ABB RAPID module: P702.mod

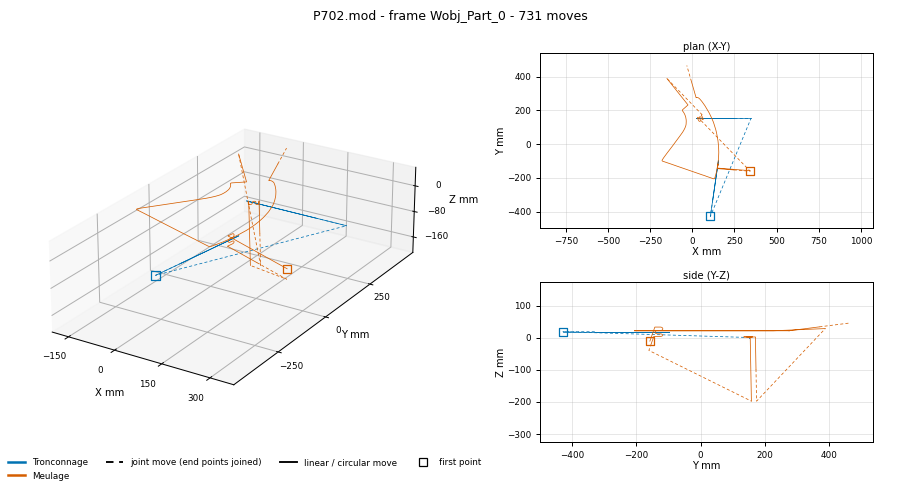
[picture p0: tool path of P702.mod in frame Wobj_Part_0, 731 of 741 moves have a stored position in this frame; points joined in program order, loops and branches not executed]
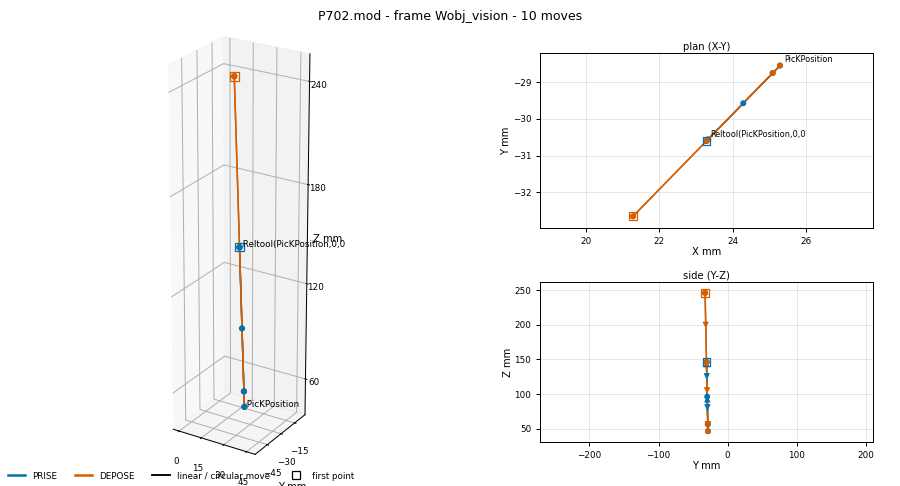
[picture p1: tool path of P702.mod in frame Wobj_vision, 10 of 741 moves have a stored position in this frame; points joined in program order, loops and branches not executed]
MODULE P702

    ! Nom         :P702
    ! Description :
    ! Créé le     :26/05/2023 11:39:24

    LOCAL CONST SPEEDDATA VitesseLente :=[10,500,0,0];
	LOCAL CONST SPEEDDATA VitesseRapide :=[30,500,0,0];
	LOCAL CONST SPEEDDATA VitesseTronconnage :=[2,500,0,0];
	LOCAL CONST SPEEDDATA VitesseTronconnageApp :=[10,500,0,0];
    !
    !Point de prise
    LOCAL PERS Robtarget PicKPosition := [[25.2898814792726,-28.5440039905978,46.3111401766051],[0.0100988844033144,-0.999721568162291,-0.0187160658859885,-0.0102228940466498],[0,0,0,0],[8.999999E+09,8.999999E+09,8.999999E+09,8.999999E+09,8.999999E+09,8.999999E+09]];
	LOCAL PERS Pose Ref := [[0,0,0],[1,0,0,0]];
    !
    !Declaration des points de meulage

    !Tr_meulage_motif_1 : Meulage d'un motif
    LOCAL CONST Robtarget Tr_meulage_motif_1_0 := [[148.038015625,-142.293734375,33.02674609375],[0.573441761718492,-0.459065341021942,-0.424059487360605,0.529714177428792],[0,0,0,0],[8.999999E+09,8.999999E+09,8.999999E+09,8.999999E+09,8.999999E+09,8.999999E+09]];
    LOCAL CONST Robtarget Tr_meulage_motif_1_1 := [[148.1818125,-141.304125,33.02651953125],[0.573441761718492,-0.459065341021942,-0.424059487360605,0.529714177428792],[0,0,0,0],[8.999999E+09,8.999999E+09,8.999999E+09,8.999999E+09,8.999999E+09,8.999999E+09]];
    LOCAL CONST Robtarget Tr_meulage_motif_1_2 := [[148.325609375,-140.314515625,33.0262890625],[0.573441761718492,-0.459065341021942,-0.424059487360605,0.529714177428792],[0,0,0,0],[8.999999E+09,8.999999E+09,8.999999E+09,8.999999E+09,8.999999E+09,8.999999E+09]];
    LOCAL CONST Robtarget Tr_meulage_motif_1_3 := [[148.46940625,-139.32490625,33.02605859375],[0.573441761718492,-0.459065341021942,-0.424059487360605,0.529714177428792],[0,0,0,0],[8.999999E+09,8.999999E+09,8.999999E+09,8.999999E+09,8.999999E+09,8.999999E+09]];
    LOCAL CONST Robtarget Tr_meulage_motif_1_4 := [[148.613203125,-138.335296875,33.025828125],[0.573441761718492,-0.459065341021942,-0.424059487360605,0.529714177428792],[0,0,0,0],[8.999999E+09,8.999999E+09,8.999999E+09,8.999999E+09,8.999999E+09,8.999999E+09]];
    LOCAL CONST Robtarget Tr_meulage_motif_1_5 := [[148.757,-137.3456875,33.02559765625],[0.573441761718492,-0.459065341021942,-0.424059487360605,0.529714177428792],[0,0,0,0],[8.999999E+09,8.999999E+09,8.999999E+09,8.999999E+09,8.999999E+09,8.999999E+09]];
    LOCAL CONST Robtarget Tr_meulage_motif_1_6 := [[148.900796875,-136.35609375,33.0253671875],[0.573441761718492,-0.459065341021942,-0.424059487360605,0.529714177428792],[0,0,0,0],[8.999999E+09,8.999999E+09,8.999999E+09,8.999999E+09,8.999999E+09,8.999999E+09]];
    LOCAL CONST Robtarget Tr_meulage_motif_1_7 := [[149.04459375,-135.366484375,33.02513671875],[0.573441761718492,-0.459065341021942,-0.424059487360605,0.529714177428792],[0,0,0,0],[8.999999E+09,8.999999E+09,8.999999E+09,8.999999E+09,8.999999E+09,8.999999E+09]];
    LOCAL CONST Robtarget Tr_meulage_motif_1_8 := [[149.188390625,-134.376875,33.02490625],[0.573441761718492,-0.459065341021942,-0.424059487360605,0.529714177428792],[0,0,0,0],[8.999999E+09,8.999999E+09,8.999999E+09,8.999999E+09,8.999999E+09,8.999999E+09]];
    LOCAL CONST Robtarget Tr_meulage_motif_1_9 := [[149.3321875,-133.387265625,33.02467578125],[0.573441761718492,-0.459065341021942,-0.424059487360605,0.529714177428792],[0,0,0,0],[8.999999E+09,8.999999E+09,8.999999E+09,8.999999E+09,8.999999E+09,8.999999E+09]];
    LOCAL CONST Robtarget Tr_meulage_motif_1_10 := [[149.475984375,-132.39765625,33.0244453125],[0.573441761718492,-0.459065341021942,-0.424059487360605,0.529714177428792],[0,0,0,0],[8.999999E+09,8.999999E+09,8.999999E+09,8.999999E+09,8.999999E+09,8.999999E+09]];
    LOCAL CONST Robtarget Tr_meulage_motif_1_11 := [[149.61978125,-131.408046875,33.02421484375],[0.573441761718492,-0.459065341021942,-0.424059487360605,0.529714177428792],[0,0,0,0],[8.999999E+09,8.999999E+09,8.999999E+09,8.999999E+09,8.999999E+09,8.999999E+09]];
    LOCAL CONST Robtarget Tr_meulage_motif_1_12 := [[149.763578125,-130.4184453125,33.023984375],[0.573441761718492,-0.459065341021942,-0.424059487360605,0.529714177428792],[0,0,0,0],[8.999999E+09,8.999999E+09,8.999999E+09,8.999999E+09,8.999999E+09,8.999999E+09]];
    LOCAL CONST Robtarget Tr_meulage_motif_1_13 := [[149.907375,-129.4288359375,33.0237578125],[0.573441761718492,-0.459065341021942,-0.424059487360605,0.529714177428792],[0,0,0,0],[8.999999E+09,8.999999E+09,8.999999E+09,8.999999E+09,8.999999E+09,8.999999E+09]];
    LOCAL CONST Robtarget Tr_meulage_motif_1_14 := [[150.051171875,-128.4392265625,33.02352734375],[0.573441761718492,-0.459065341021942,-0.424059487360605,0.529714177428792],[0,0,0,0],[8.999999E+09,8.999999E+09,8.999999E+09,8.999999E+09,8.999999E+09,8.999999E+09]];
    LOCAL CONST Robtarget Tr_meulage_motif_1_15 := [[150.19496875,-127.449625,33.023296875],[0.573441761718492,-0.459065341021942,-0.424059487360605,0.529714177428792],[0,0,0,0],[8.999999E+09,8.999999E+09,8.999999E+09,8.999999E+09,8.999999E+09,8.999999E+09]];
    LOCAL CONST Robtarget Tr_meulage_motif_1_16 := [[150.338765625,-126.460015625,33.02306640625],[0.573441761718492,-0.459065341021942,-0.424059487360605,0.529714177428792],[0,0,0,0],[8.999999E+09,8.999999E+09,8.999999E+09,8.999999E+09,8.999999E+09,8.999999E+09]];
    LOCAL CONST Robtarget Tr_meulage_motif_1_17 := [[150.4825625,-125.47040625,33.0228359375],[0.573441761718492,-0.459065341021942,-0.424059487360605,0.529714177428792],[0,0,0,0],[8.999999E+09,8.999999E+09,8.999999E+09,8.999999E+09,8.999999E+09,8.999999E+09]];
    LOCAL CONST Robtarget Tr_meulage_motif_1_18 := [[150.626359375,-124.480796875,33.02260546875],[0.573441761718492,-0.459065341021942,-0.424059487360605,0.529714177428792],[0,0,0,0],[8.999999E+09,8.999999E+09,8.999999E+09,8.999999E+09,8.999999E+09,8.999999E+09]];
    LOCAL CONST Robtarget Tr_meulage_motif_1_19 := [[150.7724375,-123.4990703125,32.9118359375],[0.573441761718492,-0.459065341021942,-0.424059487360605,0.529714177428792],[0,0,0,0],[8.999999E+09,8.999999E+09,8.999999E+09,8.999999E+09,8.999999E+09,8.999999E+09]];
    LOCAL CONST Robtarget Tr_meulage_motif_1_20 := [[150.914953125,-122.5633828125,32.700529296875],[0.573441761718492,-0.459065341021942,-0.424059487360605,0.529714177428792],[0,0,0,0],[8.999999E+09,8.999999E+09,8.999999E+09,8.999999E+09,8.999999E+09,8.999999E+09]];
    LOCAL CONST Robtarget Tr_meulage_motif_1_21 := [[151.045796875,-121.7207890625,32.4286171875],[0.573441761718492,-0.459065341021942,-0.424059487360605,0.529714177428792],[0,0,0,0],[8.999999E+09,8.999999E+09,8.999999E+09,8.999999E+09,8.999999E+09,8.999999E+09]];
    LOCAL CONST Robtarget Tr_meulage_motif_1_22 := [[151.162,-120.979921875,32.15263671875],[0.573441761718492,-0.459065341021942,-0.424059487360605,0.529714177428792],[0,0,0,0],[8.999999E+09,8.999999E+09,8.999999E+09,8.999999E+09,8.999999E+09,8.999999E+09]];
    LOCAL CONST Robtarget Tr_meulage_motif_1_23 := [[151.339015625,-119.89315625,31.536548828125],[0.573441761718492,-0.459065341021942,-0.424059487360605,0.529714177428792],[0,0,0,0],[8.999999E+09,8.999999E+09,8.999999E+09,8.999999E+09,8.999999E+09,8.999999E+09]];
    LOCAL CONST Robtarget Tr_meulage_motif_1_24 := [[151.5119375,-118.883859375,30.6890546875],[0.573441761718492,-0.459065341021942,-0.424059487360605,0.529714177428792],[0,0,0,0],[8.999999E+09,8.999999E+09,8.999999E+09,8.999999E+09,8.999999E+09,8.999999E+09]];
    LOCAL CONST Robtarget Tr_meulage_motif_1_25 := [[151.664859375,-118.0497578125,29.665466796875],[0.573441761718492,-0.459065341021942,-0.424059487360605,0.529714177428792],[0,0,0,0],[8.999999E+09,8.999999E+09,8.999999E+09,8.999999E+09,8.999999E+09,8.999999E+09]];
    LOCAL CONST Robtarget Tr_meulage_motif_1_26 := [[151.768890625,-117.5718515625,28.54969140625],[0.573441761718492,-0.459065341021942,-0.424059487360605,0.529714177428792],[0,0,0,0],[8.999999E+09,8.999999E+09,8.999999E+09,8.999999E+09,8.999999E+09,8.999999E+09]];
    LOCAL CONST Robtarget Tr_meulage_motif_1_27 := [[151.793875,-117.548296875,27.85404296875],[0.573441761718492,-0.459065341021942,-0.424059487360605,0.529714177428792],[0,0,0,0],[8.999999E+09,8.999999E+09,8.999999E+09,8.999999E+09,8.999999E+09,8.999999E+09]];
    LOCAL CONST Robtarget Tr_meulage_motif_1_28 := [[151.813921875,-117.551359375,27.193103515625],[0.573441761718492,-0.459065341021942,-0.424059487360605,0.529714177428792],[0,0,0,0],[8.999999E+09,8.999999E+09,8.999999E+09,8.999999E+09,8.999999E+09,8.999999E+09]];
    LOCAL CONST Robtarget Tr_meulage_motif_1_29 := [[151.8260625,-117.608734375,26.532333984375],[0.573441761718492,-0.459065341021942,-0.424059487360605,0.529714177428792],[0,0,0,0],[8.999999E+09,8.999999E+09,8.999999E+09,8.999999E+09,8.999999E+09,8.999999E+09]];
    LOCAL CONST Robtarget Tr_meulage_motif_1_30 := [[151.7878125,-118.1068828125,25.431216796875],[0.573441761718492,-0.459065341021942,-0.424059487360605,0.529714177428792],[0,0,0,0],[8.999999E+09,8.999999E+09,8.999999E+09,8.999999E+09,8.999999E+09,8.999999E+09]];
    LOCAL CONST Robtarget Tr_meulage_motif_1_31 := [[151.695140625,-118.9592734375,24.42526171875],[0.573441761718492,-0.459065341021942,-0.424059487360605,0.529714177428792],[0,0,0,0],[8.999999E+09,8.999999E+09,8.999999E+09,8.999999E+09,8.999999E+09,8.999999E+09]];
    LOCAL CONST Robtarget Tr_meulage_motif_1_32 := [[151.573109375,-119.9758828125,23.59701171875],[0.573441761718492,-0.459065341021942,-0.424059487360605,0.529714177428792],[0,0,0,0],[8.999999E+09,8.999999E+09,8.999999E+09,8.999999E+09,8.999999E+09,8.999999E+09]];
    LOCAL CONST Robtarget Tr_meulage_motif_1_33 := [[151.486296875,-120.657671875,23.201607421875],[0.573441761718492,-0.459065341021942,-0.424059487360605,0.529714177428792],[0,0,0,0],[8.999999E+09,8.999999E+09,8.999999E+09,8.999999E+09,8.999999E+09,8.999999E+09]];
    LOCAL CONST Robtarget Tr_meulage_motif_1_34 := [[151.33453125,-121.8060546875,22.714572265625],[0.573441761718492,-0.459065341021942,-0.424059487360605,0.529714177428792],[0,0,0,0],[8.999999E+09,8.999999E+09,8.999999E+09,8.999999E+09,8.999999E+09,8.999999E+09]];
    LOCAL CONST Robtarget Tr_meulage_motif_1_35 := [[151.22103125,-122.6435234375,22.450796875],[0.573441761718492,-0.459065341021942,-0.424059487360605,0.529714177428792],[0,0,0,0],[8.999999E+09,8.999999E+09,8.999999E+09,8.999999E+09,8.999999E+09,8.999999E+09]];
    LOCAL CONST Robtarget Tr_meulage_motif_1_36 := [[151.093203125,-123.5667890625,22.246638671875],[0.573441761718492,-0.459065341021942,-0.424059487360605,0.529714177428792],[0,0,0,0],[8.999999E+09,8.999999E+09,8.999999E+09,8.999999E+09,8.999999E+09,8.999999E+09]];
    LOCAL CONST Robtarget Tr_meulage_motif_1_37 := [[150.955359375,-124.53865625,22.138322265625],[0.573441761718492,-0.459065341021942,-0.424059487360605,0.529714177428792],[0,0,0,0],[8.999999E+09,8.999999E+09,8.999999E+09,8.999999E+09,8.999999E+09,8.999999E+09]];
    LOCAL CONST Robtarget Tr_meulage_motif_1_38 := [[150.815984375,-125.5214140625,22.0280078125],[0.573441761718492,-0.459065341021942,-0.424059487360605,0.529714177428792],[0,0,0,0],[8.999999E+09,8.999999E+09,8.999999E+09,8.999999E+09,8.999999E+09,8.999999E+09]];
    LOCAL CONST Robtarget Tr_meulage_motif_1_39 := [[150.6721875,-126.511015625,22.02823828125],[0.573441761718492,-0.459065341021942,-0.424059487360605,0.529714177428792],[0,0,0,0],[8.999999E+09,8.999999E+09,8.999999E+09,8.999999E+09,8.999999E+09,8.999999E+09]];
    LOCAL CONST Robtarget Tr_meulage_motif_1_40 := [[150.528390625,-127.500625,22.02846875],[0.573441761718492,-0.459065341021942,-0.424059487360605,0.529714177428792],[0,0,0,0],[8.999999E+09,8.999999E+09,8.999999E+09,8.999999E+09,8.999999E+09,8.999999E+09]];
    LOCAL CONST Robtarget Tr_meulage_motif_1_41 := [[150.38459375,-128.490234375,22.02869921875],[0.573441761718492,-0.459065341021942,-0.424059487360605,0.529714177428792],[0,0,0,0],[8.999999E+09,8.999999E+09,8.999999E+09,8.999999E+09,8.999999E+09,8.999999E+09]];
    LOCAL CONST Robtarget Tr_meulage_motif_1_42 := [[150.240796875,-129.47984375,22.028927734375],[0.573441761718492,-0.459065341021942,-0.424059487360605,0.529714177428792],[0,0,0,0],[8.999999E+09,8.999999E+09,8.999999E+09,8.999999E+09,8.999999E+09,8.999999E+09]];
    LOCAL CONST Robtarget Tr_meulage_motif_1_43 := [[150.097,-130.4694453125,22.029158203125],[0.573441761718492,-0.459065341021942,-0.424059487360605,0.529714177428792],[0,0,0,0],[8.999999E+09,8.999999E+09,8.999999E+09,8.999999E+09,8.999999E+09,8.999999E+09]];
    LOCAL CONST Robtarget Tr_meulage_motif_1_44 := [[149.953203125,-131.4590625,22.029388671875],[0.573441761718492,-0.459065341021942,-0.424059487360605,0.529714177428792],[0,0,0,0],[8.999999E+09,8.999999E+09,8.999999E+09,8.999999E+09,8.999999E+09,8.999999E+09]];
    LOCAL CONST Robtarget Tr_meulage_motif_1_45 := [[149.80940625,-132.44865625,22.029619140625],[0.573441761718492,-0.459065341021942,-0.424059487360605,0.529714177428792],[0,0,0,0],[8.999999E+09,8.999999E+09,8.999999E+09,8.999999E+09,8.999999E+09,8.999999E+09]];
    LOCAL CONST Robtarget Tr_meulage_motif_1_46 := [[149.665609375,-133.438265625,22.029849609375],[0.573441761718492,-0.459065341021942,-0.424059487360605,0.529714177428792],[0,0,0,0],[8.999999E+09,8.999999E+09,8.999999E+09,8.999999E+09,8.999999E+09,8.999999E+09]];
    LOCAL CONST Robtarget Tr_meulage_motif_1_47 := [[149.5218125,-134.427875,22.030080078125],[0.573441761718492,-0.459065341021942,-0.424059487360605,0.529714177428792],[0,0,0,0],[8.999999E+09,8.999999E+09,8.999999E+09,8.999999E+09,8.999999E+09,8.999999E+09]];
    LOCAL CONST Robtarget Tr_meulage_motif_1_48 := [[149.378015625,-135.417484375,22.03030859375],[0.573441761718492,-0.459065341021942,-0.424059487360605,0.529714177428792],[0,0,0,0],[8.999999E+09,8.999999E+09,8.999999E+09,8.999999E+09,8.999999E+09,8.999999E+09]];
    LOCAL CONST Robtarget Tr_meulage_motif_1_49 := [[149.238640625,-136.40025,21.91999609375],[0.573441761718492,-0.459065341021942,-0.424059487360605,0.529714177428792],[0,0,0,0],[8.999999E+09,8.999999E+09,8.999999E+09,8.999999E+09,8.999999E+09,8.999999E+09]];
    LOCAL CONST Robtarget Tr_meulage_motif_1_50 := [[149.1089375,-137.337890625,21.709125],[0.573441761718492,-0.459065341021942,-0.424059487360605,0.529714177428792],[0,0,0,0],[8.999999E+09,8.999999E+09,8.999999E+09,8.999999E+09,8.999999E+09,8.999999E+09]];
    LOCAL CONST Robtarget Tr_meulage_motif_1_51 := [[148.994546875,-138.183,21.43760546875],[0.573441761718492,-0.459065341021942,-0.424059487360605,0.529714177428792],[0,0,0,0],[8.999999E+09,8.999999E+09,8.999999E+09,8.999999E+09,8.999999E+09,8.999999E+09]];
    LOCAL CONST Robtarget Tr_meulage_motif_1_52 := [[148.90146875,-138.888515625,21.133755859375],[0.573441761718492,-0.459065341021942,-0.424059487360605,0.529714177428792],[0,0,0,0],[8.999999E+09,8.999999E+09,8.999999E+09,8.999999E+09,8.999999E+09,8.999999E+09]];
    LOCAL CONST Robtarget Tr_meulage_motif_1_53 := [[148.772796875,-139.9153125,20.471775390625],[0.573441761718492,-0.459065341021942,-0.424059487360605,0.529714177428792],[0,0,0,0],[8.999999E+09,8.999999E+09,8.999999E+09,8.999999E+09,8.999999E+09,8.999999E+09]];
    LOCAL CONST Robtarget Tr_meulage_motif_1_54 := [[148.6704375,-140.8120625,19.57046875],[0.573441761718492,-0.459065341021942,-0.424059487360605,0.529714177428792],[0,0,0,0],[8.999999E+09,8.999999E+09,8.999999E+09,8.999999E+09,8.999999E+09,8.999999E+09]];
    LOCAL CONST Robtarget Tr_meulage_motif_1_55 := [[148.62521875,-141.3463125,18.525052734375],[0.573441761718492,-0.459065341021942,-0.424059487360605,0.529714177428792],[0,0,0,0],[8.999999E+09,8.999999E+09,8.999999E+09,8.999999E+09,8.999999E+09,8.999999E+09]];
    LOCAL CONST Robtarget Tr_meulage_motif_1_56 := [[148.61965625,-141.532390625,17.832203125],[0.573441761718492,-0.459065341021942,-0.424059487360605,0.529714177428792],[0,0,0,0],[8.999999E+09,8.999999E+09,8.999999E+09,8.999999E+09,8.999999E+09,8.999999E+09]];
    LOCAL CONST Robtarget Tr_meulage_motif_1_57 := [[148.6338125,-141.599140625,17.062580078125],[0.573441761718492,-0.459065341021942,-0.424059487360605,0.529714177428792],[0,0,0,0],[8.999999E+09,8.999999E+09,8.999999E+09,8.999999E+09,8.999999E+09,8.999999E+09]];
    LOCAL CONST Robtarget Tr_meulage_motif_1_58 := [[148.666765625,-141.53646875,16.29305078125],[0.573441761718492,-0.459065341021942,-0.424059487360605,0.529714177428792],[0,0,0,0],[8.999999E+09,8.999999E+09,8.999999E+09,8.999999E+09,8.999999E+09,8.999999E+09]];
    LOCAL CONST Robtarget Tr_meulage_motif_1_59 := [[148.760703125,-141.126375,15.1852255859375],[0.573441761718492,-0.459065341021942,-0.424059487360605,0.529714177428792],[0,0,0,0],[8.999999E+09,8.999999E+09,8.999999E+09,8.999999E+09,8.999999E+09,8.999999E+09]];
    LOCAL CONST Robtarget Tr_meulage_motif_1_60 := [[148.83803125,-140.719078125,14.5997177734375],[0.573441761718492,-0.459065341021942,-0.424059487360605,0.529714177428792],[0,0,0,0],[8.999999E+09,8.999999E+09,8.999999E+09,8.999999E+09,8.999999E+09,8.999999E+09]];
    LOCAL CONST Robtarget Tr_meulage_motif_1_61 := [[148.992484375,-139.845296875,13.7128056640625],[0.573441761718492,-0.459065341021942,-0.424059487360605,0.529714177428792],[0,0,0,0],[8.999999E+09,8.999999E+09,8.999999E+09,8.999999E+09,8.999999E+09,8.999999E+09]];
    LOCAL CONST Robtarget Tr_meulage_motif_1_62 := [[149.089265625,-139.267609375,13.2985537109375],[0.573441761718492,-0.459065341021942,-0.424059487360605,0.529714177428792],[0,0,0,0],[8.999999E+09,8.999999E+09,8.999999E+09,8.999999E+09,8.999999E+09,8.999999E+09]];
    LOCAL CONST Robtarget Tr_meulage_motif_1_63 := [[149.2665,-138.16384375,12.7544580078125],[0.573441761718492,-0.459065341021942,-0.424059487360605,0.529714177428792],[0,0,0,0],[8.999999E+09,8.999999E+09,8.999999E+09,8.999999E+09,8.999999E+09,8.999999E+09]];
    LOCAL CONST Robtarget Tr_meulage_motif_1_64 := [[149.3941875,-137.348203125,12.4589072265625],[0.573441761718492,-0.459065341021942,-0.424059487360605,0.529714177428792],[0,0,0,0],[8.999999E+09,8.999999E+09,8.999999E+09,8.999999E+09,8.999999E+09,8.999999E+09]];
    LOCAL CONST Robtarget Tr_meulage_motif_1_65 := [[149.534390625,-136.42684375,12.2543203125],[0.573441761718492,-0.459065341021942,-0.424059487360605,0.529714177428792],[0,0,0,0],[8.999999E+09,8.999999E+09,8.999999E+09,8.999999E+09,8.999999E+09,8.999999E+09]];
    LOCAL CONST Robtarget Tr_meulage_motif_1_66 := [[149.678828125,-135.455984375,12.1455517578125],[0.573441761718492,-0.459065341021942,-0.424059487360605,0.529714177428792],[0,0,0,0],[8.999999E+09,8.999999E+09,8.999999E+09,8.999999E+09,8.999999E+09,8.999999E+09]];
    LOCAL CONST Robtarget Tr_meulage_motif_1_67 := [[149.82490625,-134.47425,12.03478125],[0.573441761718492,-0.459065341021942,-0.424059487360605,0.529714177428792],[0,0,0,0],[8.999999E+09,8.999999E+09,8.999999E+09,8.999999E+09,8.999999E+09,8.999999E+09]];
    LOCAL CONST Robtarget Tr_meulage_motif_1_68 := [[149.968703125,-133.484640625,12.0345517578125],[0.573441761718492,-0.459065341021942,-0.424059487360605,0.529714177428792],[0,0,0,0],[8.999999E+09,8.999999E+09,8.999999E+09,8.999999E+09,8.999999E+09,8.999999E+09]];
    LOCAL CONST Robtarget Tr_meulage_motif_1_69 := [[150.1125,-132.49503125,12.0343212890625],[0.573441761718492,-0.459065341021942,-0.424059487360605,0.529714177428792],[0,0,0,0],[8.999999E+09,8.999999E+09,8.999999E+09,8.999999E+09,8.999999E+09,8.999999E+09]];
    LOCAL CONST Robtarget Tr_meulage_motif_1_70 := [[150.256296875,-131.505421875,12.0340908203125],[0.573441761718492,-0.459065341021942,-0.424059487360605,0.529714177428792],[0,0,0,0],[8.999999E+09,8.999999E+09,8.999999E+09,8.999999E+09,8.999999E+09,8.999999E+09]];
    LOCAL CONST Robtarget Tr_meulage_motif_1_71 := [[150.40009375,-130.5158125,12.033861328125],[0.573441761718492,-0.459065341021942,-0.424059487360605,0.529714177428792],[0,0,0,0],[8.999999E+09,8.999999E+09,8.999999E+09,8.999999E+09,8.999999E+09,8.999999E+09]];
    LOCAL CONST Robtarget Tr_meulage_motif_1_72 := [[150.543890625,-129.5262109375,12.033630859375],[0.573441761718492,-0.459065341021942,-0.424059487360605,0.529714177428792],[0,0,0,0],[8.999999E+09,8.999999E+09,8.999999E+09,8.999999E+09,8.999999E+09,8.999999E+09]];
    LOCAL CONST Robtarget Tr_meulage_motif_1_73 := [[150.6876875,-128.5366015625,12.033400390625],[0.573441761718492,-0.459065341021942,-0.424059487360605,0.529714177428792],[0,0,0,0],[8.999999E+09,8.999999E+09,8.999999E+09,8.999999E+09,8.999999E+09,8.999999E+09]];
    LOCAL CONST Robtarget Tr_meulage_motif_1_74 := [[150.831484375,-127.5469921875,12.0331708984375],[0.573441761718492,-0.459065341021942,-0.424059487360605,0.529714177428792],[0,0,0,0],[8.999999E+09,8.999999E+09,8.999999E+09,8.999999E+09,8.999999E+09,8.999999E+09]];
    LOCAL CONST Robtarget Tr_meulage_motif_1_75 := [[150.97528125,-126.557390625,12.0329404296875],[0.573441761718492,-0.459065341021942,-0.424059487360605,0.529714177428792],[0,0,0,0],[8.999999E+09,8.999999E+09,8.999999E+09,8.999999E+09,8.999999E+09,8.999999E+09]];
    LOCAL CONST Robtarget Tr_meulage_motif_1_76 := [[151.119078125,-125.56778125,12.0327099609375],[0.573441761718492,-0.459065341021942,-0.424059487360605,0.529714177428792],[0,0,0,0],[8.999999E+09,8.999999E+09,8.999999E+09,8.999999E+09,8.999999E+09,8.999999E+09]];
    LOCAL CONST Robtarget Tr_meulage_motif_1_77 := [[151.262875,-124.578171875,12.03248046875],[0.573441761718492,-0.459065341021942,-0.424059487360605,0.529714177428792],[0,0,0,0],[8.999999E+09,8.999999E+09,8.999999E+09,8.999999E+09,8.999999E+09,8.999999E+09]];
    LOCAL CONST Robtarget Tr_meulage_motif_1_78 := [[151.40896875,-123.5964375,11.9217099609375],[0.573441761718492,-0.459065341021942,-0.424059487360605,0.529714177428792],[0,0,0,0],[8.999999E+09,8.999999E+09,8.999999E+09,8.999999E+09,8.999999E+09,8.999999E+09]];
    LOCAL CONST Robtarget Tr_meulage_motif_1_79 := [[151.55146875,-122.6607578125,11.710404296875],[0.573441761718492,-0.459065341021942,-0.424059487360605,0.529714177428792],[0,0,0,0],[8.999999E+09,8.999999E+09,8.999999E+09,8.999999E+09,8.999999E+09,8.999999E+09]];
    LOCAL CONST Robtarget Tr_meulage_motif_1_80 := [[151.682328125,-121.81815625,11.4384921875],[0.573441761718492,-0.459065341021942,-0.424059487360605,0.529714177428792],[0,0,0,0],[8.999999E+09,8.999999E+09,8.999999E+09,8.999999E+09,8.999999E+09,8.999999E+09]];
    LOCAL CONST Robtarget Tr_meulage_motif_1_81 := [[151.79853125,-121.077296875,11.16251171875],[0.573441761718492,-0.459065341021942,-0.424059487360605,0.529714177428792],[0,0,0,0],[8.999999E+09,8.999999E+09,8.999999E+09,8.999999E+09,8.999999E+09,8.999999E+09]];
    LOCAL CONST Robtarget Tr_meulage_motif_1_82 := [[151.97553125,-119.99053125,10.5464228515625],[0.573441761718492,-0.459065341021942,-0.424059487360605,0.529714177428792],[0,0,0,0],[8.999999E+09,8.999999E+09,8.999999E+09,8.999999E+09,8.999999E+09,8.999999E+09]];
    LOCAL CONST Robtarget Tr_meulage_motif_1_83 := [[152.140203125,-119.0478984375,9.652654296875],[0.573441761718492,-0.459065341021942,-0.424059487360605,0.529714177428792],[0,0,0,0],[8.999999E+09,8.999999E+09,8.999999E+09,8.999999E+09,8.999999E+09,8.999999E+09]];
    LOCAL CONST Robtarget Tr_meulage_motif_1_84 := [[152.260703125,-118.450140625,8.5670244140625],[0.573441761718492,-0.459065341021942,-0.424059487360605,0.529714177428792],[0,0,0,0],[8.999999E+09,8.999999E+09,8.999999E+09,8.999999E+09,8.999999E+09,8.999999E+09]];
    LOCAL CONST Robtarget Tr_meulage_motif_1_85 := [[152.314890625,-118.28715625,7.58307373046875],[0.573441761718492,-0.459065341021942,-0.424059487360605,0.529714177428792],[0,0,0,0],[8.999999E+09,8.999999E+09,8.999999E+09,8.999999E+09,8.999999E+09,8.999999E+09]];
    LOCAL CONST Robtarget Tr_meulage_motif_1_86 := [[152.3021875,-118.418203125,7.3785439453125],[0.573441761718492,-0.459065341021942,-0.424059487360605,0.529714177428792],[0,0,0,0],[8.999999E+09,8.999999E+09,8.999999E+09,8.999999E+09,8.999999E+09,8.999999E+09]];
    LOCAL CONST Robtarget Tr_meulage_motif_1_87 := [[152.30646875,-118.5436640625,6.6525078125],[0.573441761718492,-0.459065341021942,-0.424059487360605,0.529714177428792],[0,0,0,0],[8.999999E+09,8.999999E+09,8.999999E+09,8.999999E+09,8.999999E+09,8.999999E+09]];
    LOCAL CONST Robtarget Tr_meulage_motif_1_88 := [[152.236515625,-119.2248984375,5.71619921875],[0.573441761718492,-0.459065341021942,-0.424059487360605,0.529714177428792],[0,0,0,0],[8.999999E+09,8.999999E+09,8.999999E+09,8.999999E+09,8.999999E+09,8.999999E+09]];
    LOCAL CONST Robtarget Tr_meulage_motif_1_89 := [[152.170375,-119.7788828125,5.2527333984375],[0.573441761718492,-0.459065341021942,-0.424059487360605,0.529714177428792],[0,0,0,0],[8.999999E+09,8.999999E+09,8.999999E+09,8.999999E+09,8.999999E+09,8.999999E+09]];
    LOCAL CONST Robtarget Tr_meulage_motif_1_90 := [[152.023921875,-120.89990625,4.72280517578125],[0.573441761718492,-0.459065341021942,-0.424059487360605,0.529714177428792],[0,0,0,0],[8.999999E+09,8.999999E+09,8.999999E+09,8.999999E+09,8.999999E+09,8.999999E+09]];
    LOCAL CONST Robtarget Tr_meulage_motif_1_91 := [[151.910421875,-121.7373828125,4.4590302734375],[0.573441761718492,-0.459065341021942,-0.424059487360605,0.529714177428792],[0,0,0,0],[8.999999E+09,8.999999E+09,8.999999E+09,8.999999E+09,8.999999E+09,8.999999E+09]];
    LOCAL CONST Robtarget Tr_meulage_motif_1_92 := [[151.78259375,-122.660640625,4.2548720703125],[0.573441761718492,-0.459065341021942,-0.424059487360605,0.529714177428792],[0,0,0,0],[8.999999E+09,8.999999E+09,8.999999E+09,8.999999E+09,8.999999E+09,8.999999E+09]];
    LOCAL CONST Robtarget Tr_meulage_motif_1_93 := [[151.644734375,-123.6325078125,4.14655517578125],[0.573441761718492,-0.459065341021942,-0.424059487360605,0.529714177428792],[0,0,0,0],[8.999999E+09,8.999999E+09,8.999999E+09,8.999999E+09,8.999999E+09,8.999999E+09]];
    LOCAL CONST Robtarget Tr_meulage_motif_1_94 := [[151.505359375,-124.615265625,4.03624194335938],[0.573441761718492,-0.459065341021942,-0.424059487360605,0.529714177428792],[0,0,0,0],[8.999999E+09,8.999999E+09,8.999999E+09,8.999999E+09,8.999999E+09,8.999999E+09]];
    LOCAL CONST Robtarget Tr_meulage_motif_1_95 := [[151.3615625,-125.604875,4.03647216796875],[0.573441761718492,-0.459065341021942,-0.424059487360605,0.529714177428792],[0,0,0,0],[8.999999E+09,8.999999E+09,8.999999E+09,8.999999E+09,8.999999E+09,8.999999E+09]];
    LOCAL CONST Robtarget Tr_meulage_motif_1_96 := [[151.217765625,-126.594484375,4.0367021484375],[0.573441761718492,-0.459065341021942,-0.424059487360605,0.529714177428792],[0,0,0,0],[8.999999E+09,8.999999E+09,8.999999E+09,8.999999E+09,8.999999E+09,8.999999E+09]];
    LOCAL CONST Robtarget Tr_meulage_motif_1_97 := [[151.07396875,-127.5840859375,4.03693237304688],[0.573441761718492,-0.459065341021942,-0.424059487360605,0.529714177428792],[0,0,0,0],[8.999999E+09,8.999999E+09,8.999999E+09,8.999999E+09,8.999999E+09,8.999999E+09]];
    LOCAL CONST Robtarget Tr_meulage_motif_1_98 := [[150.930171875,-128.5736953125,4.03716259765625],[0.573441761718492,-0.459065341021942,-0.424059487360605,0.529714177428792],[0,0,0,0],[8.999999E+09,8.999999E+09,8.999999E+09,8.999999E+09,8.999999E+09,8.999999E+09]];
    LOCAL CONST Robtarget Tr_meulage_motif_1_99 := [[150.786375,-129.5633046875,4.037392578125],[0.573441761718492,-0.459065341021942,-0.424059487360605,0.529714177428792],[0,0,0,0],[8.999999E+09,8.999999E+09,8.999999E+09,8.999999E+09,8.999999E+09,8.999999E+09]];
    LOCAL CONST Robtarget Tr_meulage_motif_1_100 := [[150.642578125,-130.5529140625,4.03762280273437],[0.573441761718492,-0.459065341021942,-0.424059487360605,0.529714177428792],[0,0,0,0],[8.999999E+09,8.999999E+09,8.999999E+09,8.999999E+09,8.999999E+09,8.999999E+09]];
    LOCAL CONST Robtarget Tr_meulage_motif_1_101 := [[150.49878125,-131.542515625,4.03785278320313],[0.573441761718492,-0.459065341021942,-0.424059487360605,0.529714177428792],[0,0,0,0],[8.999999E+09,8.999999E+09,8.999999E+09,8.999999E+09,8.999999E+09,8.999999E+09]];
    LOCAL CONST Robtarget Tr_meulage_motif_1_102 := [[150.354984375,-132.532125,4.0380830078125],[0.573441761718492,-0.459065341021942,-0.424059487360605,0.529714177428792],[0,0,0,0],[8.999999E+09,8.999999E+09,8.999999E+09,8.999999E+09,8.999999E+09,8.999999E+09]];
    LOCAL CONST Robtarget Tr_meulage_motif_1_103 := [[150.2111875,-133.521734375,4.03831323242188],[0.573441761718492,-0.459065341021942,-0.424059487360605,0.529714177428792],[0,0,0,0],[8.999999E+09,8.999999E+09,8.999999E+09,8.999999E+09,8.999999E+09,8.999999E+09]];
    LOCAL CONST Robtarget Tr_meulage_motif_1_104 := [[150.067390625,-134.51134375,4.03854321289062],[0.573441761718492,-0.459065341021942,-0.424059487360605,0.529714177428792],[0,0,0,0],[8.999999E+09,8.999999E+09,8.999999E+09,8.999999E+09,8.999999E+09,8.999999E+09]];
    LOCAL CONST Robtarget Tr_meulage_motif_1_105 := [[149.92359375,-135.500953125,4.0387734375],[0.573441761718492,-0.459065341021942,-0.424059487360605,0.529714177428792],[0,0,0,0],[8.999999E+09,8.999999E+09,8.999999E+09,8.999999E+09,8.999999E+09,8.999999E+09]];
    LOCAL CONST Robtarget Tr_meulage_motif_1_106 := [[149.779796875,-136.490546875,4.03900366210938],[0.573441761718492,-0.459065341021942,-0.424059487360605,0.529714177428792],[0,0,0,0],[8.999999E+09,8.999999E+09,8.999999E+09,8.999999E+09,8.999999E+09,8.999999E+09]];
    LOCAL CONST Robtarget Tr_meulage_motif_1_107 := [[149.636,-137.48015625,4.03923364257813],[0.573441761718492,-0.459065341021942,-0.424059487360605,0.529714177428792],[0,0,0,0],[8.999999E+09,8.999999E+09,8.999999E+09,8.999999E+09,8.999999E+09,8.999999E+09]];
    LOCAL CONST Robtarget Tr_meulage_motif_1_108 := [[149.492203125,-138.469765625,4.0394638671875],[0.573441761718492,-0.459065341021942,-0.424059487360605,0.529714177428792],[0,0,0,0],[8.999999E+09,8.999999E+09,8.999999E+09,8.999999E+09,8.999999E+09,8.999999E+09]];
    LOCAL CONST Robtarget Tr_meulage_motif_1_109 := [[149.34840625,-139.459375,4.03969384765625],[0.573441761718492,-0.459065341021942,-0.424059487360605,0.529714177428792],[0,0,0,0],[8.999999E+09,8.999999E+09,8.999999E+09,8.999999E+09,8.999999E+09,8.999999E+09]];
    LOCAL CONST Robtarget Tr_meulage_motif_1_110 := [[149.204609375,-140.448984375,4.03992407226562],[0.573441761718492,-0.459065341021942,-0.424059487360605,0.529714177428792],[0,0,0,0],[8.999999E+09,8.999999E+09,8.999999E+09,8.999999E+09,8.999999E+09,8.999999E+09]];
    LOCAL CONST Robtarget Tr_meulage_motif_1_111 := [[149.0608125,-141.43859375,4.040154296875],[0.573441761718492,-0.459065341021942,-0.424059487360605,0.529714177428792],[0,0,0,0],[8.999999E+09,8.999999E+09,8.999999E+09,8.999999E+09,8.999999E+09,8.999999E+09]];
    LOCAL CONST Robtarget Tr_meulage_motif_1_112 := [[148.917015625,-142.428203125,4.04038427734375],[0.573441761718492,-0.459065341021942,-0.424059487360605,0.529714177428792],[0,0,0,0],[8.999999E+09,8.999999E+09,8.999999E+09,8.999999E+09,8.999999E+09,8.999999E+09]];
    LOCAL CONST Robtarget Tr_meulage_motif_1_113 := [[148.77321875,-143.417796875,4.04061450195312],[0.573441761718492,-0.459065341021942,-0.424059487360605,0.529714177428792],[0,0,0,0],[8.999999E+09,8.999999E+09,8.999999E+09,8.999999E+09,8.999999E+09,8.999999E+09]];
    LOCAL CONST Robtarget Tr_meulage_motif_1_114 := [[148.629421875,-144.40740625,4.0408447265625],[0.573441761718492,-0.459065341021942,-0.424059487360605,0.529714177428792],[0,0,0,0],[8.999999E+09,8.999999E+09,8.999999E+09,8.999999E+09,8.999999E+09,8.999999E+09]];
    LOCAL CONST Robtarget Tr_meulage_motif_1_115 := [[148.485625,-145.397015625,4.04107470703125],[0.573441761718492,-0.459065341021942,-0.424059487360605,0.529714177428792],[0,0,0,0],[8.999999E+09,8.999999E+09,8.999999E+09,8.999999E+09,8.999999E+09,8.999999E+09]];

    !Tr_meulage_motif_2 : Meulage d'un motif
    LOCAL CONST Robtarget Tr_meulage_motif_2_0 := [[29.6025625,154.628359375,2.27771118164063],[8.63642748194515E-05,0.00936471427117237,0.00922151094472952,-0.999913625471584],[0,0,0,0],[8.999999E+09,8.999999E+09,8.999999E+09,8.999999E+09,8.999999E+09,8.999999E+09]];
    LOCAL CONST Robtarget Tr_meulage_motif_2_1 := [[30.06765234375,153.74309375,2.28043334960938],[8.63642748194515E-05,0.00936471427117237,0.00922151094472952,-0.999913625471584],[0,0,0,0],[8.999999E+09,8.999999E+09,8.999999E+09,8.999999E+09,8.999999E+09,8.999999E+09]];
    LOCAL CONST Robtarget Tr_meulage_motif_2_2 := [[30.5327421875,152.857828125,2.28315551757813],[8.63642748194515E-05,0.00936471427117237,0.00922151094472952,-0.999913625471584],[0,0,0,0],[8.999999E+09,8.999999E+09,8.999999E+09,8.999999E+09,8.999999E+09,8.999999E+09]];
    LOCAL CONST Robtarget Tr_meulage_motif_2_3 := [[30.99783203125,151.972578125,2.2858779296875],[8.63642748194515E-05,0.00936471427117237,0.00922151094472952,-0.999913625471584],[0,0,0,0],[8.999999E+09,8.999999E+09,8.999999E+09,8.999999E+09,8.999999E+09,8.999999E+09]];
    LOCAL CONST Robtarget Tr_meulage_motif_2_4 := [[31.462919921875,151.0873125,2.28860009765625],[8.63642748194515E-05,0.00936471427117237,0.00922151094472952,-0.999913625471584],[0,0,0,0],[8.999999E+09,8.999999E+09,8.999999E+09,8.999999E+09,8.999999E+09,8.999999E+09]];
    LOCAL CONST Robtarget Tr_meulage_motif_2_5 := [[31.928009765625,150.2020625,2.291322265625],[8.63642748194515E-05,0.00936471427117237,0.00922151094472952,-0.999913625471584],[0,0,0,0],[8.999999E+09,8.999999E+09,8.999999E+09,8.999999E+09,8.999999E+09,8.999999E+09]];
    LOCAL CONST Robtarget Tr_meulage_motif_2_6 := [[32.393099609375,149.316796875,2.29404467773438],[8.63642748194515E-05,0.00936471427117237,0.00922151094472952,-0.999913625471584],[0,0,0,0],[8.999999E+09,8.999999E+09,8.999999E+09,8.999999E+09,8.999999E+09,8.999999E+09]];
    LOCAL CONST Robtarget Tr_meulage_motif_2_7 := [[32.8581875,148.43153125,2.29676684570313],[8.63642748194515E-05,0.00936471427117237,0.00922151094472952,-0.999913625471584],[0,0,0,0],[8.999999E+09,8.999999E+09,8.999999E+09,8.999999E+09,8.999999E+09,8.999999E+09]];
    LOCAL CONST Robtarget Tr_meulage_motif_2_8 := [[33.32327734375,147.54628125,2.2994892578125],[8.63642748194515E-05,0.00936471427117237,0.00922151094472952,-0.999913625471584],[0,0,0,0],[8.999999E+09,8.999999E+09,8.999999E+09,8.999999E+09,8.999999E+09,8.999999E+09]];
    LOCAL CONST Robtarget Tr_meulage_motif_2_9 := [[33.7883671875,146.661015625,2.30221142578125],[8.63642748194515E-05,0.00936471427117237,0.00922151094472952,-0.999913625471584],[0,0,0,0],[8.999999E+09,8.999999E+09,8.999999E+09,8.999999E+09,8.999999E+09,8.999999E+09]];
    LOCAL CONST Robtarget Tr_meulage_motif_2_10 := [[34.25345703125,145.77575,2.30493359375],[8.63642748194515E-05,0.00936471427117237,0.00922151094472952,-0.999913625471584],[0,0,0,0],[8.999999E+09,8.999999E+09,8.999999E+09,8.999999E+09,8.999999E+09,8.999999E+09]];
    LOCAL CONST Robtarget Tr_meulage_motif_2_11 := [[34.718546875,144.8905,2.30765600585937],[8.63642748194515E-05,0.00936471427117237,0.00922151094472952,-0.999913625471584],[0,0,0,0],[8.999999E+09,8.999999E+09,8.999999E+09,8.999999E+09,8.999999E+09,8.999999E+09]];
    LOCAL CONST Robtarget Tr_meulage_motif_2_12 := [[35.18363671875,144.005234375,2.31037817382813],[8.63642748194515E-05,0.00936471427117237,0.00922151094472952,-0.999913625471584],[0,0,0,0],[8.999999E+09,8.999999E+09,8.999999E+09,8.999999E+09,8.999999E+09,8.999999E+09]];
    LOCAL CONST Robtarget Tr_meulage_motif_2_13 := [[35.6487265625,143.119984375,2.31310034179688],[8.63642748194515E-05,0.00936471427117237,0.00922151094472952,-0.999913625471584],[0,0,0,0],[8.999999E+09,8.999999E+09,8.999999E+09,8.999999E+09,8.999999E+09,8.999999E+09]];
    LOCAL CONST Robtarget Tr_meulage_motif_2_14 := [[36.11381640625,142.23471875,2.31582275390625],[8.63642748194515E-05,0.00936471427117237,0.00922151094472952,-0.999913625471584],[0,0,0,0],[8.999999E+09,8.999999E+09,8.999999E+09,8.999999E+09,8.999999E+09,8.999999E+09]];
    LOCAL CONST Robtarget Tr_meulage_motif_2_15 := [[36.57890625,141.349453125,2.318544921875],[8.63642748194515E-05,0.00936471427117237,0.00922151094472952,-0.999913625471584],[0,0,0,0],[8.999999E+09,8.999999E+09,8.999999E+09,8.999999E+09,8.999999E+09,8.999999E+09]];
    LOCAL CONST Robtarget Tr_meulage_motif_2_16 := [[37.0439921875,140.464203125,2.32126708984375],[8.63642748194515E-05,0.00936471427117237,0.00922151094472952,-0.999913625471584],[0,0,0,0],[8.999999E+09,8.999999E+09,8.999999E+09,8.999999E+09,8.999999E+09,8.999999E+09]];
    LOCAL CONST Robtarget Tr_meulage_motif_2_17 := [[37.50908203125,139.5789375,2.32398950195312],[8.63642748194515E-05,0.00936471427117237,0.00922151094472952,-0.999913625471584],[0,0,0,0],[8.999999E+09,8.999999E+09,8.999999E+09,8.999999E+09,8.999999E+09,8.999999E+09]];
    LOCAL CONST Robtarget Tr_meulage_motif_2_18 := [[37.974171875,138.6936875,2.32671166992187],[8.63642748194515E-05,0.00936471427117237,0.00922151094472952,-0.999913625471584],[0,0,0,0],[8.999999E+09,8.999999E+09,8.999999E+09,8.999999E+09,8.999999E+09,8.999999E+09]];
    LOCAL CONST Robtarget Tr_meulage_motif_2_19 := [[38.53370703125,137.8664375,2.32925048828125],[8.63642748194515E-05,0.00936471427117237,0.00922151094472952,-0.999913625471584],[0,0,0,0],[8.999999E+09,8.999999E+09,8.999999E+09,8.999999E+09,8.999999E+09,8.999999E+09]];
    LOCAL CONST Robtarget Tr_meulage_motif_2_20 := [[39.16087109375,137.126765625,2.33151586914063],[8.63642748194515E-05,0.00936471427117237,0.00922151094472952,-0.999913625471584],[0,0,0,0],[8.999999E+09,8.999999E+09,8.999999E+09,8.999999E+09,8.999999E+09,8.999999E+09]];
    LOCAL CONST Robtarget Tr_meulage_motif_2_21 := [[39.79811328125,136.4983125,2.33343627929688],[8.63642748194515E-05,0.00936471427117237,0.00922151094472952,-0.999913625471584],[0,0,0,0],[8.999999E+09,8.999999E+09,8.999999E+09,8.999999E+09,8.999999E+09,8.999999E+09]];
    LOCAL CONST Robtarget Tr_meulage_motif_2_22 := [[40.3911796875,135.962765625,2.33507104492188],[8.63642748194515E-05,0.00936471427117237,0.00922151094472952,-0.999913625471584],[0,0,0,0],[8.999999E+09,8.999999E+09,8.999999E+09,8.999999E+09,8.999999E+09,8.999999E+09]];
    LOCAL CONST Robtarget Tr_meulage_motif_2_23 := [[41.44870703125,135.27459375,2.33715991210937],[8.63642748194515E-05,0.00936471427117237,0.00922151094472952,-0.999913625471584],[0,0,0,0],[8.999999E+09,8.999999E+09,8.999999E+09,8.999999E+09,8.999999E+09,8.999999E+09]];
    LOCAL CONST Robtarget Tr_meulage_motif_2_24 := [[42.67530078125,134.762421875,2.338697265625],[8.63642748194515E-05,0.00936471427117237,0.00922151094472952,-0.999913625471584],[0,0,0,0],[8.999999E+09,8.999999E+09,8.999999E+09,8.999999E+09,8.999999E+09,8.999999E+09]];
    LOCAL CONST Robtarget Tr_meulage_motif_2_25 := [[43.97593359375,134.48821875,2.3394951171875],[8.63642748194515E-05,0.00936471427117237,0.00922151094472952,-0.999913625471584],[0,0,0,0],[8.999999E+09,8.999999E+09,8.999999E+09,8.999999E+09,8.999999E+09,8.999999E+09]];
    LOCAL CONST Robtarget Tr_meulage_motif_2_26 := [[45.19108984375,134.575203125,2.33917822265625],[8.63642748194515E-05,0.00936471427117237,0.00922151094472952,-0.999913625471584],[0,0,0,0],[8.999999E+09,8.999999E+09,8.999999E+09,8.999999E+09,8.999999E+09,8.999999E+09]];
    LOCAL CONST Robtarget Tr_meulage_motif_2_27 := [[45.81979296875,134.8749375,2.3382255859375],[8.63642748194515E-05,0.00936471427117237,0.00922151094472952,-0.999913625471584],[0,0,0,0],[8.999999E+09,8.999999E+09,8.999999E+09,8.999999E+09,8.999999E+09,8.999999E+09]];
    LOCAL CONST Robtarget Tr_meulage_motif_2_28 := [[46.40517578125,135.18246875,2.33725048828125],[8.63642748194515E-05,0.00936471427117237,0.00922151094472952,-0.999913625471584],[0,0,0,0],[8.999999E+09,8.999999E+09,8.999999E+09,8.999999E+09,8.999999E+09,8.999999E+09]];
    LOCAL CONST Robtarget Tr_meulage_motif_2_29 := [[46.96489453125,135.538515625,2.33612646484375],[8.63642748194515E-05,0.00936471427117237,0.00922151094472952,-0.999913625471584],[0,0,0,0],[8.999999E+09,8.999999E+09,8.999999E+09,8.999999E+09,8.999999E+09,8.999999E+09]];
    LOCAL CONST Robtarget Tr_meulage_motif_2_30 := [[47.708515625,136.491984375,2.33314575195313],[8.63642748194515E-05,0.00936471427117237,0.00922151094472952,-0.999913625471584],[0,0,0,0],[8.999999E+09,8.999999E+09,8.999999E+09,8.999999E+09,8.999999E+09,8.999999E+09]];
    LOCAL CONST Robtarget Tr_meulage_motif_2_31 := [[48.20123828125,137.718484375,2.32932934570313],[8.63642748194515E-05,0.00936471427117237,0.00922151094472952,-0.999913625471584],[0,0,0,0],[8.999999E+09,8.999999E+09,8.999999E+09,8.999999E+09,8.999999E+09,8.999999E+09]];
    LOCAL CONST Robtarget Tr_meulage_motif_2_32 := [[48.45903515625,139.009953125,2.3253212890625],[8.63642748194515E-05,0.00936471427117237,0.00922151094472952,-0.999913625471584],[0,0,0,0],[8.999999E+09,8.999999E+09,8.999999E+09,8.999999E+09,8.999999E+09,8.999999E+09]];
    LOCAL CONST Robtarget Tr_meulage_motif_2_33 := [[48.4898203125,139.80228125,2.32286743164063],[8.63642748194515E-05,0.00936471427117237,0.00922151094472952,-0.999913625471584],[0,0,0,0],[8.999999E+09,8.999999E+09,8.999999E+09,8.999999E+09,8.999999E+09,8.999999E+09]];
    LOCAL CONST Robtarget Tr_meulage_motif_2_34 := [[48.382765625,141.05428125,2.31899560546875],[8.63642748194515E-05,0.00936471427117237,0.00922151094472952,-0.999913625471584],[0,0,0,0],[8.999999E+09,8.999999E+09,8.999999E+09,8.999999E+09,8.999999E+09,8.999999E+09]];
    LOCAL CONST Robtarget Tr_meulage_motif_2_35 := [[48.22354296875,141.9251875,2.31630590820312],[8.63642748194515E-05,0.00936471427117237,0.00922151094472952,-0.999913625471584],[0,0,0,0],[8.999999E+09,8.999999E+09,8.999999E+09,8.999999E+09,8.999999E+09,8.999999E+09]];
    LOCAL CONST Robtarget Tr_meulage_motif_2_36 := [[47.97108984375,142.84534375,2.31346728515625],[8.63642748194515E-05,0.00936471427117237,0.00922151094472952,-0.999913625471584],[0,0,0,0],[8.999999E+09,8.999999E+09,8.999999E+09,8.999999E+09,8.999999E+09,8.999999E+09]];
    LOCAL CONST Robtarget Tr_meulage_motif_2_37 := [[47.6107109375,143.76478125,2.31063500976563],[8.63642748194515E-05,0.00936471427117237,0.00922151094472952,-0.999913625471584],[0,0,0,0],[8.999999E+09,8.999999E+09,8.999999E+09,8.999999E+09,8.999999E+09,8.999999E+09]];
    LOCAL CONST Robtarget Tr_meulage_motif_2_38 := [[47.246984375,144.69490625,2.30777001953125],[8.63642748194515E-05,0.00936471427117237,0.00922151094472952,-0.999913625471584],[0,0,0,0],[8.999999E+09,8.999999E+09,8.999999E+09,8.999999E+09,8.999999E+09,8.999999E+09]];
    LOCAL CONST Robtarget Tr_meulage_motif_2_39 := [[46.78189453125,145.58015625,2.3050478515625],[8.63642748194515E-05,0.00936471427117237,0.00922151094472952,-0.999913625471584],[0,0,0,0],[8.999999E+09,8.999999E+09,8.999999E+09,8.999999E+09,8.999999E+09,8.999999E+09]];
    LOCAL CONST Robtarget Tr_meulage_motif_2_40 := [[46.3168046875,146.465421875,2.30232543945313],[8.63642748194515E-05,0.00936471427117237,0.00922151094472952,-0.999913625471584],[0,0,0,0],[8.999999E+09,8.999999E+09,8.999999E+09,8.999999E+09,8.999999E+09,8.999999E+09]];
    LOCAL CONST Robtarget Tr_meulage_motif_2_41 := [[45.85171484375,147.350671875,2.29960327148438],[8.63642748194515E-05,0.00936471427117237,0.00922151094472952,-0.999913625471584],[0,0,0,0],[8.999999E+09,8.999999E+09,8.999999E+09,8.999999E+09,8.999999E+09,8.999999E+09]];
    LOCAL CONST Robtarget Tr_meulage_motif_2_42 := [[45.386625,148.2359375,2.29688110351562],[8.63642748194515E-05,0.00936471427117237,0.00922151094472952,-0.999913625471584],[0,0,0,0],[8.999999E+09,8.999999E+09,8.999999E+09,8.999999E+09,8.999999E+09,8.999999E+09]];
    LOCAL CONST Robtarget Tr_meulage_motif_2_43 := [[44.92153515625,149.121203125,2.29415869140625],[8.63642748194515E-05,0.00936471427117237,0.00922151094472952,-0.999913625471584],[0,0,0,0],[8.999999E+09,8.999999E+09,8.999999E+09,8.999999E+09,8.999999E+09,8.999999E+09]];
    LOCAL CONST Robtarget Tr_meulage_motif_2_44 := [[44.45644921875,150.006453125,2.2914365234375],[8.63642748194515E-05,0.00936471427117237,0.00922151094472952,-0.999913625471584],[0,0,0,0],[8.999999E+09,8.999999E+09,8.999999E+09,8.999999E+09,8.999999E+09,8.999999E+09]];
    LOCAL CONST Robtarget Tr_meulage_motif_2_45 := [[43.991359375,150.89171875,2.28871435546875],[8.63642748194515E-05,0.00936471427117237,0.00922151094472952,-0.999913625471584],[0,0,0,0],[8.999999E+09,8.999999E+09,8.999999E+09,8.999999E+09,8.999999E+09,8.999999E+09]];
    LOCAL CONST Robtarget Tr_meulage_motif_2_46 := [[43.52626953125,151.77696875,2.28599194335938],[8.63642748194515E-05,0.00936471427117237,0.00922151094472952,-0.999913625471584],[0,0,0,0],[8.999999E+09,8.999999E+09,8.999999E+09,8.999999E+09,8.999999E+09,8.999999E+09]];
    LOCAL CONST Robtarget Tr_meulage_motif_2_47 := [[43.0611796875,152.662234375,2.28326977539063],[8.63642748194515E-05,0.00936471427117237,0.00922151094472952,-0.999913625471584],[0,0,0,0],[8.999999E+09,8.999999E+09,8.999999E+09,8.999999E+09,8.999999E+09,8.999999E+09]];
    LOCAL CONST Robtarget Tr_meulage_motif_2_48 := [[42.59608984375,153.5475,2.28054736328125],[8.63642748194515E-05,0.00936471427117237,0.00922151094472952,-0.999913625471584],[0,0,0,0],[8.999999E+09,8.999999E+09,8.999999E+09,8.999999E+09,8.999999E+09,8.999999E+09]];
    LOCAL CONST Robtarget Tr_meulage_motif_2_49 := [[42.23236328125,154.477609375,2.27768237304688],[8.63642748194515E-05,0.00936471427117237,0.00922151094472952,-0.999913625471584],[0,0,0,0],[8.999999E+09,8.999999E+09,8.999999E+09,8.999999E+09,8.999999E+09,8.999999E+09]];
    LOCAL CONST Robtarget Tr_meulage_motif_2_50 := [[41.97911328125,155.41371875,2.27479443359375],[8.63642748194515E-05,0.00936471427117237,0.00922151094472952,-0.999913625471584],[0,0,0,0],[8.999999E+09,8.999999E+09,8.999999E+09,8.999999E+09,8.999999E+09,8.999999E+09]];
    LOCAL CONST Robtarget Tr_meulage_motif_2_51 := [[41.82317578125,156.29503125,2.272072265625],[8.63642748194515E-05,0.00936471427117237,0.00922151094472952,-0.999913625471584],[0,0,0,0],[8.999999E+09,8.999999E+09,8.999999E+09,8.999999E+09,8.999999E+09,8.999999E+09]];
    LOCAL CONST Robtarget Tr_meulage_motif_2_52 := [[41.7615234375,157.066359375,2.26968701171875],[8.63642748194515E-05,0.00936471427117237,0.00922151094472952,-0.999913625471584],[0,0,0,0],[8.999999E+09,8.999999E+09,8.999999E+09,8.999999E+09,8.999999E+09,8.999999E+09]];
    LOCAL CONST Robtarget Tr_meulage_motif_2_53 := [[41.86691796875,158.290265625,2.26589379882813],[8.63642748194515E-05,0.00936471427117237,0.00922151094472952,-0.999913625471584],[0,0,0,0],[8.999999E+09,8.999999E+09,8.999999E+09,8.999999E+09,8.999999E+09,8.999999E+09]];
    LOCAL CONST Robtarget Tr_meulage_motif_2_54 := [[42.245890625,159.5081875,2.26210864257812],[8.63642748194515E-05,0.00936471427117237,0.00922151094472952,-0.999913625471584],[0,0,0,0],[8.999999E+09,8.999999E+09,8.999999E+09,8.999999E+09,8.999999E+09,8.999999E+09]];
    LOCAL CONST Robtarget Tr_meulage_motif_2_55 := [[42.92309375,160.468265625,2.25911010742188],[8.63642748194515E-05,0.00936471427117237,0.00922151094472952,-0.999913625471584],[0,0,0,0],[8.999999E+09,8.999999E+09,8.999999E+09,8.999999E+09,8.999999E+09,8.999999E+09]];
    LOCAL CONST Robtarget Tr_meulage_motif_2_56 := [[43.4508359375,160.954265625,2.2575849609375],[8.63642748194515E-05,0.00936471427117237,0.00922151094472952,-0.999913625471584],[0,0,0,0],[8.999999E+09,8.999999E+09,8.999999E+09,8.999999E+09,8.999999E+09,8.999999E+09]];
    LOCAL CONST Robtarget Tr_meulage_motif_2_57 := [[44.102796875,161.368890625,2.25627563476562],[8.63642748194515E-05,0.00936471427117237,0.00922151094472952,-0.999913625471584],[0,0,0,0],[8.999999E+09,8.999999E+09,8.999999E+09,8.999999E+09,8.999999E+09,8.999999E+09]];
    LOCAL CONST Robtarget Tr_meulage_motif_2_58 := [[44.81546875,161.6676875,2.25532275390625],[8.63642748194515E-05,0.00936471427117237,0.00922151094472952,-0.999913625471584],[0,0,0,0],[8.999999E+09,8.999999E+09,8.999999E+09,8.999999E+09,8.999999E+09,8.999999E+09]];
    LOCAL CONST Robtarget Tr_meulage_motif_2_59 := [[45.9917109375,161.811671875,2.25483081054688],[8.63642748194515E-05,0.00936471427117237,0.00922151094472952,-0.999913625471584],[0,0,0,0],[8.999999E+09,8.999999E+09,8.999999E+09,8.999999E+09,8.999999E+09,8.999999E+09]];
    LOCAL CONST Robtarget Tr_meulage_motif_2_60 := [[46.70289453125,161.717296875,2.25509521484375],[8.63642748194515E-05,0.00936471427117237,0.00922151094472952,-0.999913625471584],[0,0,0,0],[8.999999E+09,8.999999E+09,8.999999E+09,8.999999E+09,8.999999E+09,8.999999E+09]];
    LOCAL CONST Robtarget Tr_meulage_motif_2_61 := [[47.90082421875,161.3445625,2.2562021484375],[8.63642748194515E-05,0.00936471427117237,0.00922151094472952,-0.999913625471584],[0,0,0,0],[8.999999E+09,8.999999E+09,8.999999E+09,8.999999E+09,8.999999E+09,8.999999E+09]];
    LOCAL CONST Robtarget Tr_meulage_motif_2_62 := [[48.53999609375,161.018765625,2.257185546875],[8.63642748194515E-05,0.00936471427117237,0.00922151094472952,-0.999913625471584],[0,0,0,0],[8.999999E+09,8.999999E+09,8.999999E+09,8.999999E+09,8.999999E+09,8.999999E+09]];
    LOCAL CONST Robtarget Tr_meulage_motif_2_63 := [[49.54158984375,160.282171875,2.25942651367188],[8.63642748194515E-05,0.00936471427117237,0.00922151094472952,-0.999913625471584],[0,0,0,0],[8.999999E+09,8.999999E+09,8.999999E+09,8.999999E+09,8.999999E+09,8.999999E+09]];
    LOCAL CONST Robtarget Tr_meulage_motif_2_64 := [[50.18716015625,159.68875,2.26123828125],[8.63642748194515E-05,0.00936471427117237,0.00922151094472952,-0.999913625471584],[0,0,0,0],[8.999999E+09,8.999999E+09,8.999999E+09,8.999999E+09,8.999999E+09,8.999999E+09]];
    LOCAL CONST Robtarget Tr_meulage_motif_2_65 := [[50.8016328125,158.95878125,2.26347387695313],[8.63642748194515E-05,0.00936471427117237,0.00922151094472952,-0.999913625471584],[0,0,0,0],[8.999999E+09,8.999999E+09,8.999999E+09,8.999999E+09,8.999999E+09,8.999999E+09]];
    LOCAL CONST Robtarget Tr_meulage_motif_2_66 := [[51.35428125,158.14034375,2.26598583984375],[8.63642748194515E-05,0.00936471427117237,0.00922151094472952,-0.999913625471584],[0,0,0,0],[8.999999E+09,8.999999E+09,8.999999E+09,8.999999E+09,8.999999E+09,8.999999E+09]];
    LOCAL CONST Robtarget Tr_meulage_motif_2_67 := [[51.91381640625,157.313109375,2.26852490234375],[8.63642748194515E-05,0.00936471427117237,0.00922151094472952,-0.999913625471584],[0,0,0,0],[8.999999E+09,8.999999E+09,8.999999E+09,8.999999E+09,8.999999E+09,8.999999E+09]];
    LOCAL CONST Robtarget Tr_meulage_motif_2_68 := [[52.37890625,156.42784375,2.2712470703125],[8.63642748194515E-05,0.00936471427117237,0.00922151094472952,-0.999913625471584],[0,0,0,0],[8.999999E+09,8.999999E+09,8.999999E+09,8.999999E+09,8.999999E+09,8.999999E+09]];
    LOCAL CONST Robtarget Tr_meulage_motif_2_69 := [[52.84399609375,155.54259375,2.27396923828125],[8.63642748194515E-05,0.00936471427117237,0.00922151094472952,-0.999913625471584],[0,0,0,0],[8.999999E+09,8.999999E+09,8.999999E+09,8.999999E+09,8.999999E+09,8.999999E+09]];
    LOCAL CONST Robtarget Tr_meulage_motif_2_70 := [[53.3090859375,154.657328125,2.27669165039062],[8.63642748194515E-05,0.00936471427117237,0.00922151094472952,-0.999913625471584],[0,0,0,0],[8.999999E+09,8.999999E+09,8.999999E+09,8.999999E+09,8.999999E+09,8.999999E+09]];
    LOCAL CONST Robtarget Tr_meulage_motif_2_71 := [[53.77417578125,153.7720625,2.27941381835937],[8.63642748194515E-05,0.00936471427117237,0.00922151094472952,-0.999913625471584],[0,0,0,0],[8.999999E+09,8.999999E+09,8.999999E+09,8.999999E+09,8.999999E+09,8.999999E+09]];
    LOCAL CONST Robtarget Tr_meulage_motif_2_72 := [[54.23926171875,152.8868125,2.28213598632813],[8.63642748194515E-05,0.00936471427117237,0.00922151094472952,-0.999913625471584],[0,0,0,0],[8.999999E+09,8.999999E+09,8.999999E+09,8.999999E+09,8.999999E+09,8.999999E+09]];
    LOCAL CONST Robtarget Tr_meulage_motif_2_73 := [[54.7043515625,152.001546875,2.2848583984375],[8.63642748194515E-05,0.00936471427117237,0.00922151094472952,-0.999913625471584],[0,0,0,0],[8.999999E+09,8.999999E+09,8.999999E+09,8.999999E+09,8.999999E+09,8.999999E+09]];
    LOCAL CONST Robtarget Tr_meulage_motif_2_74 := [[55.16944140625,151.11628125,2.28758056640625],[8.63642748194515E-05,0.00936471427117237,0.00922151094472952,-0.999913625471584],[0,0,0,0],[8.999999E+09,8.999999E+09,8.999999E+09,8.999999E+09,8.999999E+09,8.999999E+09]];
    LOCAL CONST Robtarget Tr_meulage_motif_2_75 := [[55.63453125,150.23103125,2.290302734375],[8.63642748194515E-05,0.00936471427117237,0.00922151094472952,-0.999913625471584],[0,0,0,0],[8.999999E+09,8.999999E+09,8.999999E+09,8.999999E+09,8.999999E+09,8.999999E+09]];
    LOCAL CONST Robtarget Tr_meulage_motif_2_76 := [[56.09962109375,149.345765625,2.29302514648437],[8.63642748194515E-05,0.00936471427117237,0.00922151094472952,-0.999913625471584],[0,0,0,0],[8.999999E+09,8.999999E+09,8.999999E+09,8.999999E+09,8.999999E+09,8.999999E+09]];
    LOCAL CONST Robtarget Tr_meulage_motif_2_77 := [[56.5647109375,148.460515625,2.29574731445312],[8.63642748194515E-05,0.00936471427117237,0.00922151094472952,-0.999913625471584],[0,0,0,0],[8.999999E+09,8.999999E+09,8.999999E+09,8.999999E+09,8.999999E+09,8.999999E+09]];
    LOCAL CONST Robtarget Tr_meulage_motif_2_78 := [[57.12424609375,147.633265625,2.29828637695313],[8.63642748194515E-05,0.00936471427117237,0.00922151094472952,-0.999913625471584],[0,0,0,0],[8.999999E+09,8.999999E+09,8.999999E+09,8.999999E+09,8.999999E+09,8.999999E+09]];
    LOCAL CONST Robtarget Tr_meulage_motif_2_79 := [[57.75141015625,146.89359375,2.30055151367187],[8.63642748194515E-05,0.00936471427117237,0.00922151094472952,-0.999913625471584],[0,0,0,0],[8.999999E+09,8.999999E+09,8.999999E+09,8.999999E+09,8.999999E+09,8.999999E+09]];
    LOCAL CONST Robtarget Tr_meulage_motif_2_80 := [[58.38865234375,146.265140625,2.30247192382813],[8.63642748194515E-05,0.00936471427117237,0.00922151094472952,-0.999913625471584],[0,0,0,0],[8.999999E+09,8.999999E+09,8.999999E+09,8.999999E+09,8.999999E+09,8.999999E+09]];
    LOCAL CONST Robtarget Tr_meulage_motif_2_81 := [[58.98171875,145.72959375,2.30410668945313],[8.63642748194515E-05,0.00936471427117237,0.00922151094472952,-0.999913625471584],[0,0,0,0],[8.999999E+09,8.999999E+09,8.999999E+09,8.999999E+09,8.999999E+09,8.999999E+09]];
    LOCAL CONST Robtarget Tr_meulage_motif_2_82 := [[60.0392421875,145.041421875,2.30619555664062],[8.63642748194515E-05,0.00936471427117237,0.00922151094472952,-0.999913625471584],[0,0,0,0],[8.999999E+09,8.999999E+09,8.999999E+09,8.999999E+09,8.999999E+09,8.999999E+09]];
    LOCAL CONST Robtarget Tr_meulage_motif_2_83 := [[61.2756015625,144.61025,2.30748168945312],[8.63642748194515E-05,0.00936471427117237,0.00922151094472952,-0.999913625471584],[0,0,0,0],[8.999999E+09,8.999999E+09,8.999999E+09,8.999999E+09,8.999999E+09,8.999999E+09]];
    LOCAL CONST Robtarget Tr_meulage_motif_2_84 := [[62.520296875,144.57609375,2.30753857421875],[8.63642748194515E-05,0.00936471427117237,0.00922151094472952,-0.999913625471584],[0,0,0,0],[8.999999E+09,8.999999E+09,8.999999E+09,8.999999E+09,8.999999E+09,8.999999E+09]];
    LOCAL CONST Robtarget Tr_meulage_motif_2_85 := [[63.47047265625,144.88403125,2.30654809570313],[8.63642748194515E-05,0.00936471427117237,0.00922151094472952,-0.999913625471584],[0,0,0,0],[8.999999E+09,8.999999E+09,8.999999E+09,8.999999E+09,8.999999E+09,8.999999E+09]];
    LOCAL CONST Robtarget Tr_meulage_motif_2_86 := [[63.59050390625,145.09559375,2.30588842773437],[8.63642748194515E-05,0.00936471427117237,0.00922151094472952,-0.999913625471584],[0,0,0,0],[8.999999E+09,8.999999E+09,8.999999E+09,8.999999E+09,8.999999E+09,8.999999E+09]];
    LOCAL CONST Robtarget Tr_meulage_motif_2_87 := [[64.17618359375,145.54265625,2.3044814453125],[8.63642748194515E-05,0.00936471427117237,0.00922151094472952,-0.999913625471584],[0,0,0,0],[8.999999E+09,8.999999E+09,8.999999E+09,8.999999E+09,8.999999E+09,8.999999E+09]];
    LOCAL CONST Robtarget Tr_meulage_motif_2_88 := [[64.68747265625,146.583921875,2.30123803710938],[8.63642748194515E-05,0.00936471427117237,0.00922151094472952,-0.999913625471584],[0,0,0,0],[8.999999E+09,8.999999E+09,8.999999E+09,8.999999E+09,8.999999E+09,8.999999E+09]];
    LOCAL CONST Robtarget Tr_meulage_motif_2_89 := [[64.83872265625,147.29328125,2.2990361328125],[8.63642748194515E-05,0.00936471427117237,0.00922151094472952,-0.999913625471584],[0,0,0,0],[8.999999E+09,8.999999E+09,8.999999E+09,8.999999E+09,8.999999E+09,8.999999E+09]];
    LOCAL CONST Robtarget Tr_meulage_motif_2_90 := [[64.7826015625,148.54059375,2.29517700195313],[8.63642748194515E-05,0.00936471427117237,0.00922151094472952,-0.999913625471584],[0,0,0,0],[8.999999E+09,8.999999E+09,8.999999E+09,8.999999E+09,8.999999E+09,8.999999E+09]];
    LOCAL CONST Robtarget Tr_meulage_motif_2_91 := [[64.62337890625,149.4115,2.2924873046875],[8.63642748194515E-05,0.00936471427117237,0.00922151094472952,-0.999913625471584],[0,0,0,0],[8.999999E+09,8.999999E+09,8.999999E+09,8.999999E+09,8.999999E+09,8.999999E+09]];
    LOCAL CONST Robtarget Tr_meulage_motif_2_92 := [[64.37092578125,150.33165625,2.28964868164062],[8.63642748194515E-05,0.00936471427117237,0.00922151094472952,-0.999913625471584],[0,0,0,0],[8.999999E+09,8.999999E+09,8.999999E+09,8.999999E+09,8.999999E+09,8.999999E+09]];
    LOCAL CONST Robtarget Tr_meulage_motif_2_93 := [[64.010546875,151.25109375,2.28681640625],[8.63642748194515E-05,0.00936471427117237,0.00922151094472952,-0.999913625471584],[0,0,0,0],[8.999999E+09,8.999999E+09,8.999999E+09,8.999999E+09,8.999999E+09,8.999999E+09]];
    LOCAL CONST Robtarget Tr_meulage_motif_2_94 := [[63.6468203125,152.181203125,2.28395141601563],[8.63642748194515E-05,0.00936471427117237,0.00922151094472952,-0.999913625471584],[0,0,0,0],[8.999999E+09,8.999999E+09,8.999999E+09,8.999999E+09,8.999999E+09,8.999999E+09]];
    LOCAL CONST Robtarget Tr_meulage_motif_2_95 := [[63.18173046875,153.06646875,2.28122924804688],[8.63642748194515E-05,0.00936471427117237,0.00922151094472952,-0.999913625471584],[0,0,0,0],[8.999999E+09,8.999999E+09,8.999999E+09,8.999999E+09,8.999999E+09,8.999999E+09]];
    LOCAL CONST Robtarget Tr_meulage_motif_2_96 := [[62.716640625,153.95171875,2.2785068359375],[8.63642748194515E-05,0.00936471427117237,0.00922151094472952,-0.999913625471584],[0,0,0,0],[8.999999E+09,8.999999E+09,8.999999E+09,8.999999E+09,8.999999E+09,8.999999E+09]];
    LOCAL CONST Robtarget Tr_meulage_motif_2_97 := [[62.25155078125,154.836984375,2.27578466796875],[8.63642748194515E-05,0.00936471427117237,0.00922151094472952,-0.999913625471584],[0,0,0,0],[8.999999E+09,8.999999E+09,8.999999E+09,8.999999E+09,8.999999E+09,8.999999E+09]];
    LOCAL CONST Robtarget Tr_meulage_motif_2_98 := [[61.7864609375,155.72225,2.2730625],[8.63642748194515E-05,0.00936471427117237,0.00922151094472952,-0.999913625471584],[0,0,0,0],[8.999999E+09,8.999999E+09,8.999999E+09,8.999999E+09,8.999999E+09,8.999999E+09]];
    LOCAL CONST Robtarget Tr_meulage_motif_2_99 := [[61.32137109375,156.6075,2.27034008789063],[8.63642748194515E-05,0.00936471427117237,0.00922151094472952,-0.999913625471584],[0,0,0,0],[8.999999E+09,8.999999E+09,8.999999E+09,8.999999E+09,8.999999E+09,8.999999E+09]];
    LOCAL CONST Robtarget Tr_meulage_motif_2_100 := [[60.85628515625,157.492765625,2.26761791992188],[8.63642748194515E-05,0.00936471427117237,0.00922151094472952,-0.999913625471584],[0,0,0,0],[8.999999E+09,8.999999E+09,8.999999E+09,8.999999E+09,8.999999E+09,8.999999E+09]];
    LOCAL CONST Robtarget Tr_meulage_motif_2_101 := [[60.3911953125,158.37803125,2.26489575195313],[8.63642748194515E-05,0.00936471427117237,0.00922151094472952,-0.999913625471584],[0,0,0,0],[8.999999E+09,8.999999E+09,8.999999E+09,8.999999E+09,8.999999E+09,8.999999E+09]];
    LOCAL CONST Robtarget Tr_meulage_motif_2_102 := [[59.92610546875,159.26328125,2.26217333984375],[8.63642748194515E-05,0.00936471427117237,0.00922151094472952,-0.999913625471584],[0,0,0,0],[8.999999E+09,8.999999E+09,8.999999E+09,8.999999E+09,8.999999E+09,8.999999E+09]];
    LOCAL CONST Robtarget Tr_meulage_motif_2_103 := [[59.461015625,160.148546875,2.259451171875],[8.63642748194515E-05,0.00936471427117237,0.00922151094472952,-0.999913625471584],[0,0,0,0],[8.999999E+09,8.999999E+09,8.999999E+09,8.999999E+09,8.999999E+09,8.999999E+09]];
    LOCAL CONST Robtarget Tr_meulage_motif_2_104 := [[58.99592578125,161.033796875,2.25672875976562],[8.63642748194515E-05,0.00936471427117237,0.00922151094472952,-0.999913625471584],[0,0,0,0],[8.999999E+09,8.999999E+09,8.999999E+09,8.999999E+09,8.999999E+09,8.999999E+09]];
    LOCAL CONST Robtarget Tr_meulage_motif_2_105 := [[58.5308359375,161.9190625,2.25400659179688],[8.63642748194515E-05,0.00936471427117237,0.00922151094472952,-0.999913625471584],[0,0,0,0],[8.999999E+09,8.999999E+09,8.999999E+09,8.999999E+09,8.999999E+09,8.999999E+09]];
    LOCAL CONST Robtarget Tr_meulage_motif_2_106 := [[58.06574609375,162.804328125,2.25128442382813],[8.63642748194515E-05,0.00936471427117237,0.00922151094472952,-0.999913625471584],[0,0,0,0],[8.999999E+09,8.999999E+09,8.999999E+09,8.999999E+09,8.999999E+09,8.999999E+09]];
    LOCAL CONST Robtarget Tr_meulage_motif_2_107 := [[57.60065625,163.689578125,2.24856201171875],[8.63642748194515E-05,0.00936471427117237,0.00922151094472952,-0.999913625471584],[0,0,0,0],[8.999999E+09,8.999999E+09,8.999999E+09,8.999999E+09,8.999999E+09,8.999999E+09]];
    LOCAL CONST Robtarget Tr_meulage_motif_2_108 := [[57.13556640625,164.57484375,2.24583984375],[8.63642748194515E-05,0.00936471427117237,0.00922151094472952,-0.999913625471584],[0,0,0,0],[8.999999E+09,8.999999E+09,8.999999E+09,8.999999E+09,8.999999E+09,8.999999E+09]];
    LOCAL CONST Robtarget Tr_meulage_motif_2_109 := [[56.67048046875,165.46009375,2.24311767578125],[8.63642748194515E-05,0.00936471427117237,0.00922151094472952,-0.999913625471584],[0,0,0,0],[8.999999E+09,8.999999E+09,8.999999E+09,8.999999E+09,8.999999E+09,8.999999E+09]];
    LOCAL CONST Robtarget Tr_meulage_motif_2_110 := [[56.205390625,166.345359375,2.24039526367187],[8.63642748194515E-05,0.00936471427117237,0.00922151094472952,-0.999913625471584],[0,0,0,0],[8.999999E+09,8.999999E+09,8.999999E+09,8.999999E+09,8.999999E+09,8.999999E+09]];
    LOCAL CONST Robtarget Tr_meulage_motif_2_111 := [[55.74030078125,167.230625,2.23767309570313],[8.63642748194515E-05,0.00936471427117237,0.00922151094472952,-0.999913625471584],[0,0,0,0],[8.999999E+09,8.999999E+09,8.999999E+09,8.999999E+09,8.999999E+09,8.999999E+09]];
    LOCAL CONST Robtarget Tr_meulage_motif_2_112 := [[55.2752109375,168.115875,2.23495092773438],[8.63642748194515E-05,0.00936471427117237,0.00922151094472952,-0.999913625471584],[0,0,0,0],[8.999999E+09,8.999999E+09,8.999999E+09,8.999999E+09,8.999999E+09,8.999999E+09]];
    LOCAL CONST Robtarget Tr_meulage_motif_2_113 := [[54.81012109375,169.001140625,2.232228515625],[8.63642748194515E-05,0.00936471427117237,0.00922151094472952,-0.999913625471584],[0,0,0,0],[8.999999E+09,8.999999E+09,8.999999E+09,8.999999E+09,8.999999E+09,8.999999E+09]];
    LOCAL CONST Robtarget Tr_meulage_motif_2_114 := [[54.34503125,169.886390625,2.22950634765625],[8.63642748194515E-05,0.00936471427117237,0.00922151094472952,-0.999913625471584],[0,0,0,0],[8.999999E+09,8.999999E+09,8.999999E+09,8.999999E+09,8.999999E+09,8.999999E+09]];
    LOCAL CONST Robtarget Tr_meulage_motif_2_115 := [[53.87994140625,170.77165625,2.2267841796875],[8.63642748194515E-05,0.00936471427117237,0.00922151094472952,-0.999913625471584],[0,0,0,0],[8.999999E+09,8.999999E+09,8.999999E+09,8.999999E+09,8.999999E+09,8.999999E+09]];

